// TIA Portal V17 export
// export: Created 2024-09-02T12:50:23.4161598Z, ExportSetting WithDefaults, DisplayName Totally Integrated Automation Portal, DisplayVersion V17, DisplayName TIA Portal Openness, DisplayVersion V17, DisplayName TIA Portal Version Control Interface, DisplayVersion V17, DisplayName STEP 7 Professional, DisplayVersion V17, DisplayName STEP 7 Safety, DisplayVersion V17, DisplayName WinCC Professional, DisplayVersion V17
FUNCTION "AnwFC_Aveva_OP702" : Void   // FC36, LAD
{ S7_Optimized_Access := 'TRUE' }
VERSION : 0.1
// stored: AutoNumber false, IsIECCheckEnabled false, SetENOAutomatically false, UDAEnableTagReadback false
   VAR_TEMP
      Data_Ready : Bool;
      Pallet_Nr_Moved : Bool;
      Converted_Data : Real;
      tEKSLevelOK : Bool;
   END_VAR
   VAR CONSTANT
      cButtonNotActive : USInt := 0;
      cButtonActive : USInt := 1;
      cColorRed : USInt := 2;
      cColorGreen : USInt := 3;
      cMesOptionEmpty : USInt := 0;
      cMesReasonEmpty : String := '';
   END_VAR
   VAR_TEMP   // added for the SCL form of the ladder/FBD networks
      _w1 : Bool;
      _w2 : Bool;
      _w3 : Bool;
      _w4 : Bool;
   END_VAR
BEGIN

REGION Network 1: ################STEP 1 - Pallet arrive to station #################
END_REGION

REGION Network 2: Copy Nr of Pallet
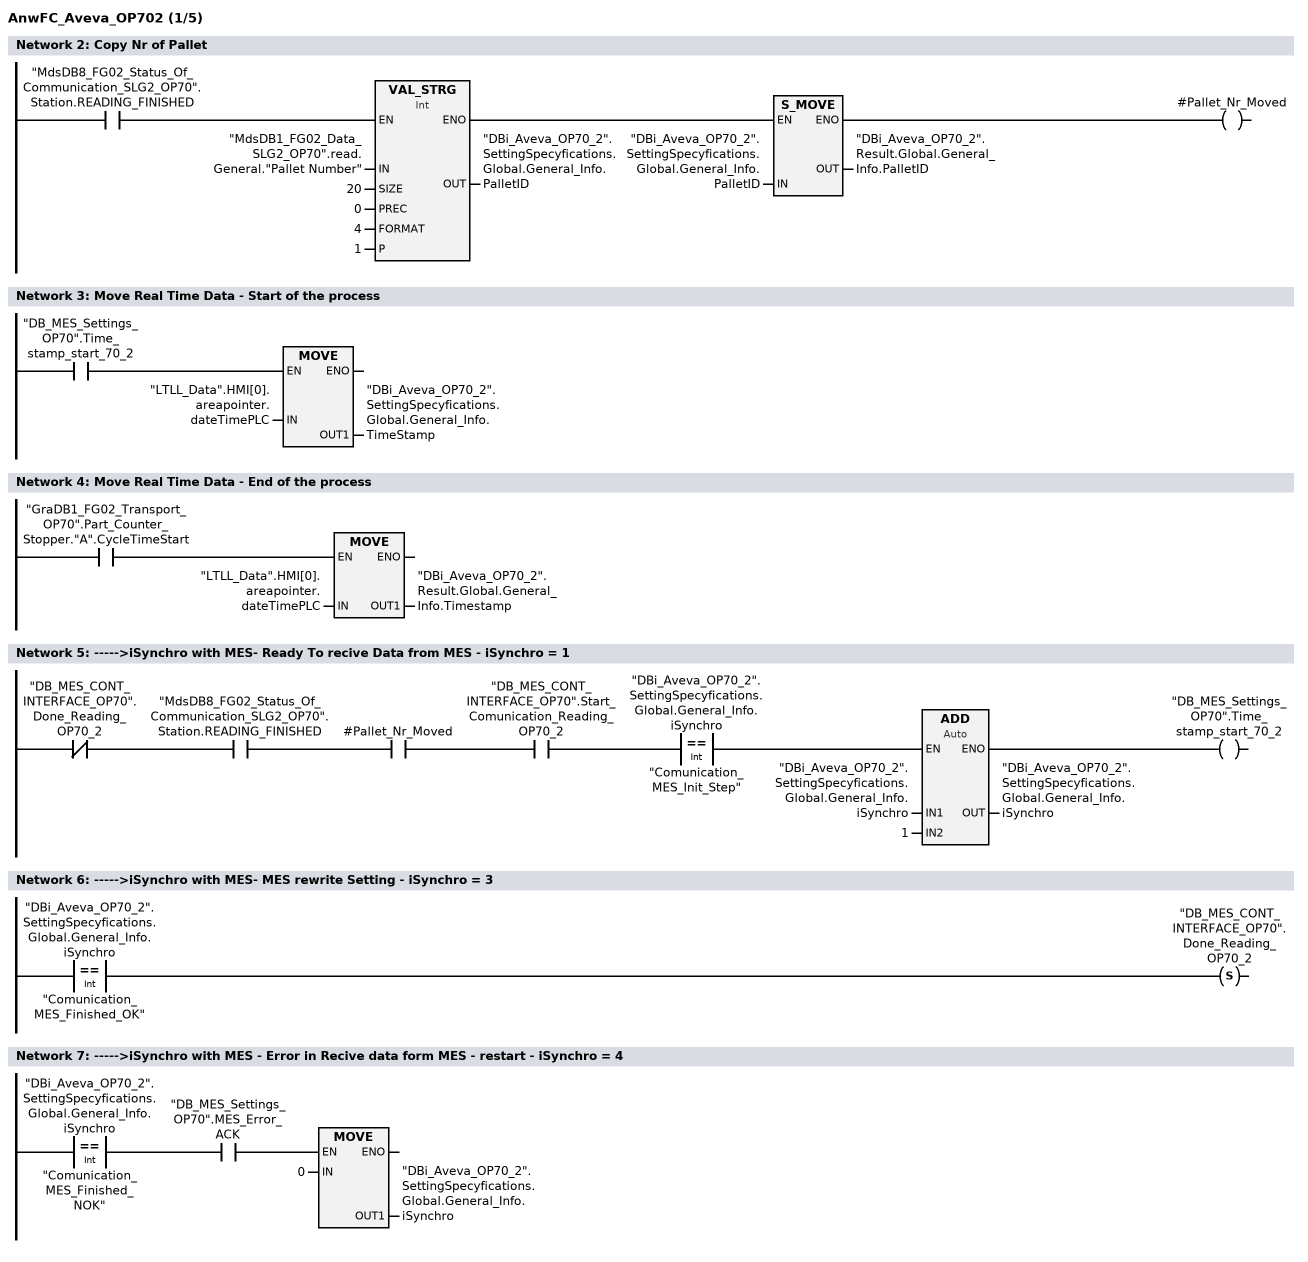
   RUNG wire#powerrail
      Contact( "MdsDB8_FG02_Status_Of_Communication_SLG2_OP70".Station.READING_FINISHED )
      { S7_Templates := "[value_type := Int, str_type := String]" } VAL_STRG(IN := "MdsDB1_FG02_Data_SLG2_OP70".read.General."Pallet Number", SIZE := 20, PREC := 0, FORMAT := 4, P := 1, OUT => "DBi_Aveva_OP70_2".SettingSpecyfications.Global.General_Info.PalletID)
      S_Move(in := "DBi_Aveva_OP70_2".SettingSpecyfications.Global.General_Info.PalletID, out => "DBi_Aveva_OP70_2".Result.Global.General_Info.PalletID)
      Coil( #Pallet_Nr_Moved )
   END_RUNG
   // the same network as SCL:
   VAL_STRG(EN := "MdsDB8_FG02_Status_Of_Communication_SLG2_OP70".Station.READING_FINISHED,
            IN := "MdsDB1_FG02_Data_SLG2_OP70".read.General."Pallet Number",
            SIZE := 20,
            PREC := 0,
            FORMAT := 4,
            P := 1,
            OUT => "DBi_Aveva_OP70_2".SettingSpecyfications.Global.General_Info.PalletID,
            ENO => #_w1);
   IF #_w1 THEN
       "DBi_Aveva_OP70_2".Result.Global.General_Info.PalletID := "DBi_Aveva_OP70_2".SettingSpecyfications.Global.General_Info.PalletID;
   END_IF;
   #Pallet_Nr_Moved := #_w1;
END_REGION

REGION Network 3: Move Real Time Data - Start of the process
   RUNG wire#powerrail
      Contact( "DB_MES_Settings_OP70".Time_stamp_start_70_2 )
      Move(in := "LTLL_Data".HMI[0].areapointer.dateTimePLC, out1 => "DBi_Aveva_OP70_2".SettingSpecyfications.Global.General_Info.TimeStamp)
   END_RUNG
   // the same network as SCL:
   IF "DB_MES_Settings_OP70".Time_stamp_start_70_2 THEN
       "DBi_Aveva_OP70_2".SettingSpecyfications.Global.General_Info.TimeStamp := "LTLL_Data".HMI[0].areapointer.dateTimePLC;
   END_IF;
END_REGION

REGION Network 4: Move Real Time Data - End of the process
   RUNG wire#powerrail
      Contact( "GraDB1_FG02_Transport_OP70".Part_Counter_Stopper."A".CycleTimeStart )
      Move(in := "LTLL_Data".HMI[0].areapointer.dateTimePLC, out1 => "DBi_Aveva_OP70_2".Result.Global.General_Info.Timestamp)
   END_RUNG
   // the same network as SCL:
   IF "GraDB1_FG02_Transport_OP70".Part_Counter_Stopper."A".CycleTimeStart THEN
       "DBi_Aveva_OP70_2".Result.Global.General_Info.Timestamp := "LTLL_Data".HMI[0].areapointer.dateTimePLC;
   END_IF;
END_REGION

REGION Network 5: ----->iSynchro with MES- Ready To recive Data from MES - iSynchro = 1
   RUNG wire#powerrail
      I_Contact( "DB_MES_CONT_INTERFACE_OP70".Done_Reading_OP70_2 )
      Contact( "MdsDB8_FG02_Status_Of_Communication_SLG2_OP70".Station.READING_FINISHED )
      Contact( #Pallet_Nr_Moved )
      Contact( "DB_MES_CONT_INTERFACE_OP70".Start_Comunication_Reading_OP70_2 )
      { S7_Templates := "SrcType := Int" } EQ_Contact(in1 := "DBi_Aveva_OP70_2".SettingSpecyfications.Global.General_Info.iSynchro, in2 := "Comunication_MES_Init_Step")
      Add(in1 := "DBi_Aveva_OP70_2".SettingSpecyfications.Global.General_Info.iSynchro, in2 := 1, out => "DBi_Aveva_OP70_2".SettingSpecyfications.Global.General_Info.iSynchro)
      Coil( "DB_MES_Settings_OP70".Time_stamp_start_70_2 )
   END_RUNG
   // the same network as SCL:
   #_w1 := NOT "DB_MES_CONT_INTERFACE_OP70".Done_Reading_OP70_2 AND "MdsDB8_FG02_Status_Of_Communication_SLG2_OP70".Station.READING_FINISHED AND #Pallet_Nr_Moved AND "DB_MES_CONT_INTERFACE_OP70".Start_Comunication_Reading_OP70_2 AND ("DBi_Aveva_OP70_2".SettingSpecyfications.Global.General_Info.iSynchro = "Comunication_MES_Init_Step");
   IF #_w1 THEN
       "DBi_Aveva_OP70_2".SettingSpecyfications.Global.General_Info.iSynchro := "DBi_Aveva_OP70_2".SettingSpecyfications.Global.General_Info.iSynchro + 1;
   END_IF;
   "DB_MES_Settings_OP70".Time_stamp_start_70_2 := #_w1;
END_REGION

REGION Network 6: ----->iSynchro with MES- MES rewrite Setting - iSynchro = 3
   RUNG wire#powerrail
      { S7_Templates := "SrcType := Int" } EQ_Contact(in1 := "DBi_Aveva_OP70_2".SettingSpecyfications.Global.General_Info.iSynchro, in2 := "Comunication_MES_Finished_OK")
      S_Coil( "DB_MES_CONT_INTERFACE_OP70".Done_Reading_OP70_2 )
   END_RUNG
   // the same network as SCL:
   IF "DBi_Aveva_OP70_2".SettingSpecyfications.Global.General_Info.iSynchro = "Comunication_MES_Finished_OK" THEN
       "DB_MES_CONT_INTERFACE_OP70".Done_Reading_OP70_2 := TRUE;
   END_IF;
END_REGION

REGION Network 7: ----->iSynchro with MES - Error in Recive data form MES - restart - iSynchro = 4
   RUNG wire#powerrail
      { S7_Templates := "SrcType := Int" } EQ_Contact(in1 := "DBi_Aveva_OP70_2".SettingSpecyfications.Global.General_Info.iSynchro, in2 := "Comunication_MES_Finished_NOK")
      Contact( "DB_MES_Settings_OP70".MES_Error_ACK )
      Move(in := 0, out1 => "DBi_Aveva_OP70_2".SettingSpecyfications.Global.General_Info.iSynchro)
   END_RUNG
   // the same network as SCL:
   IF ("DBi_Aveva_OP70_2".SettingSpecyfications.Global.General_Info.iSynchro = "Comunication_MES_Finished_NOK") AND "DB_MES_Settings_OP70".MES_Error_ACK THEN
       "DBi_Aveva_OP70_2".SettingSpecyfications.Global.General_Info.iSynchro := 0;
   END_IF;
END_REGION

REGION Network 8: ----->iSynchro with MES - End of Analyse - restart iSynchro = 0
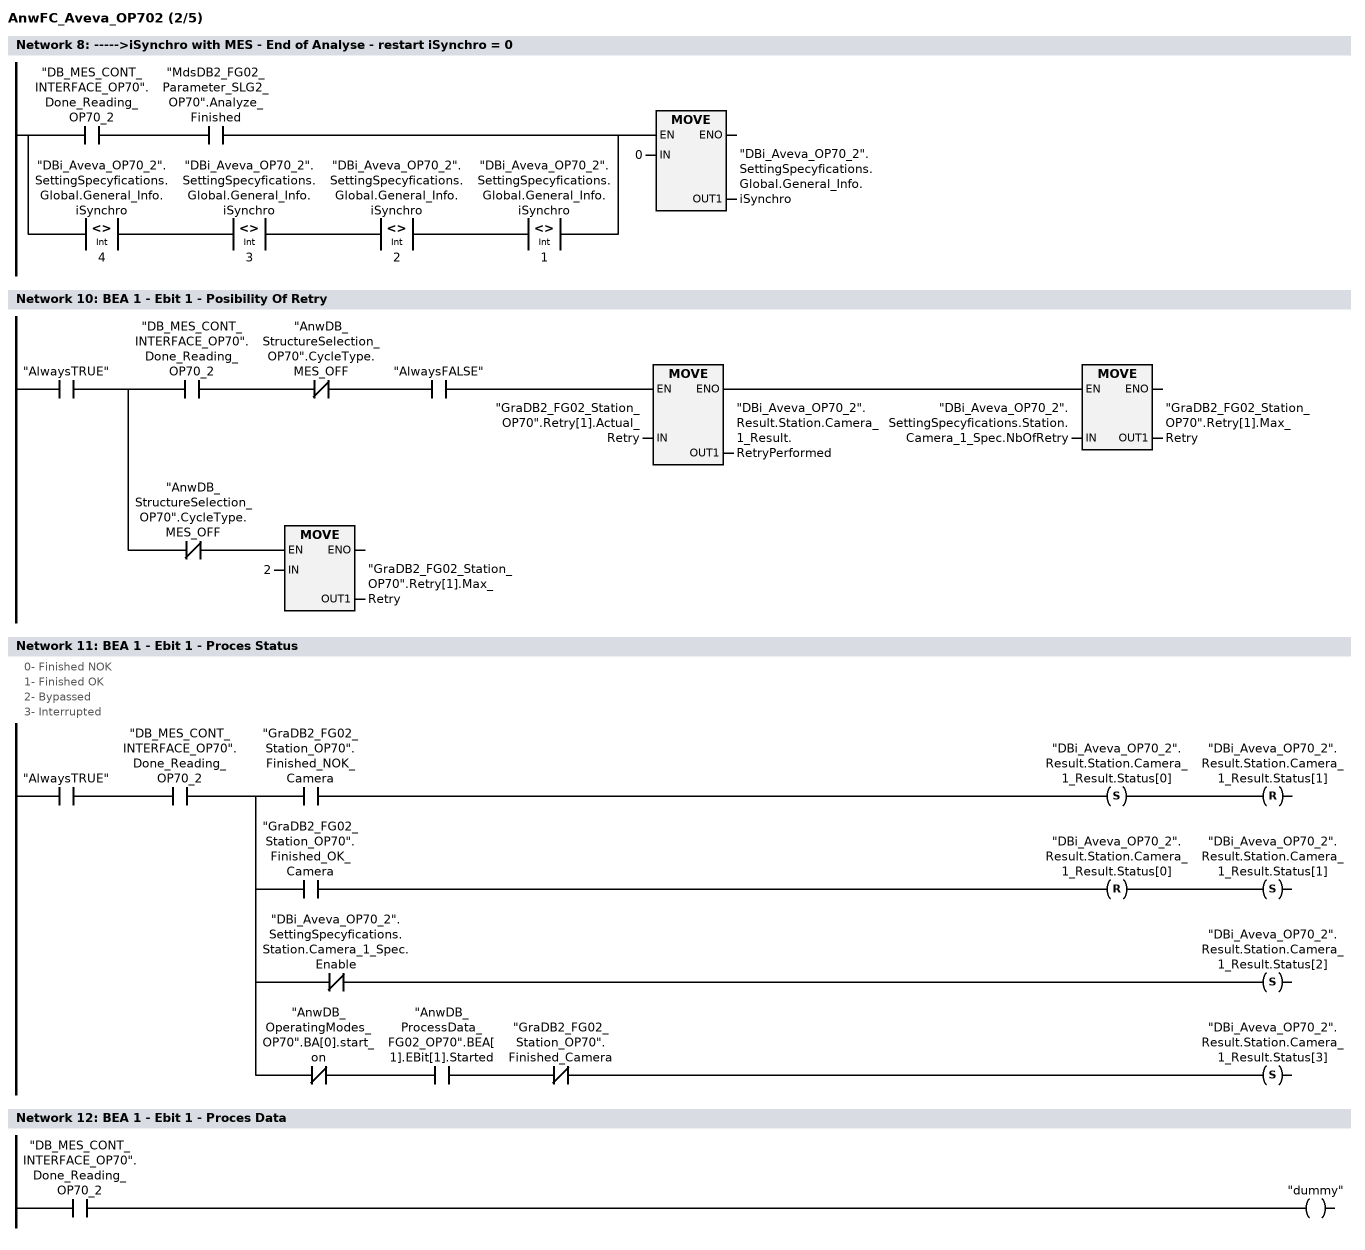
   RUNG wire#powerrail
      Contact( "DB_MES_CONT_INTERFACE_OP70".Done_Reading_OP70_2 )
      Contact( "MdsDB2_FG02_Parameter_SLG2_OP70".Analyze_Finished )
      wire#w1
      Move(in := 0, out1 => "DBi_Aveva_OP70_2".SettingSpecyfications.Global.General_Info.iSynchro)
   END_RUNG
   RUNG wire#powerrail
      { S7_Templates := "SrcType := Int" } NE_Contact(in1 := "DBi_Aveva_OP70_2".SettingSpecyfications.Global.General_Info.iSynchro, in2 := 4)
      { S7_Templates := "SrcType := Int" } NE_Contact(in1 := "DBi_Aveva_OP70_2".SettingSpecyfications.Global.General_Info.iSynchro, in2 := 3)
      { S7_Templates := "SrcType := Int" } NE_Contact(in1 := "DBi_Aveva_OP70_2".SettingSpecyfications.Global.General_Info.iSynchro, in2 := 2)
      { S7_Templates := "SrcType := Int" } NE_Contact(in1 := "DBi_Aveva_OP70_2".SettingSpecyfications.Global.General_Info.iSynchro, in2 := 1)
   END_RUNG wire#w1
   // the same network as SCL:
   IF ("DB_MES_CONT_INTERFACE_OP70".Done_Reading_OP70_2 AND "MdsDB2_FG02_Parameter_SLG2_OP70".Analyze_Finished) OR (("DBi_Aveva_OP70_2".SettingSpecyfications.Global.General_Info.iSynchro <> 4) AND ("DBi_Aveva_OP70_2".SettingSpecyfications.Global.General_Info.iSynchro <> 3) AND ("DBi_Aveva_OP70_2".SettingSpecyfications.Global.General_Info.iSynchro <> 2) AND ("DBi_Aveva_OP70_2".SettingSpecyfications.Global.General_Info.iSynchro <> 1)) THEN
       "DBi_Aveva_OP70_2".SettingSpecyfications.Global.General_Info.iSynchro := 0;
   END_IF;
END_REGION

REGION Network 9: ################STEP 2 - Move the Proce Data From Each Operation ################# / Status Proces 1
   // IN0 - Aktor ist abgewählt
   // IN1 - TAF ist angewählt
   // IN2 - Nacharbeit in Station
   // IN3 - Auftrag manuell vorgegeben
   // IN4 - Nacharbeit auf Standby-Platz
   // IN5 - Nacharbeit auf EAS-Platz
   // IN6 - TAF hat gearbeitet (Fertigmeldung)
   // IN7 - Bauteil wurde iO bearbeitet
END_REGION

REGION Network 10: BEA 1 - Ebit 1 - Posibility Of Retry
   RUNG wire#powerrail
      Contact( "AlwaysTRUE" )
      wire#w1
      Contact( "DB_MES_CONT_INTERFACE_OP70".Done_Reading_OP70_2 )
      I_Contact( "AnwDB_StructureSelection_OP70".CycleType.MES_OFF )
      Contact( "AlwaysFALSE" )
      Move(in := "GraDB2_FG02_Station_OP70".Retry[1].Actual_Retry, out1 => "DBi_Aveva_OP70_2".Result.Station.Camera_1_Result.RetryPerformed)
      Move(in := "DBi_Aveva_OP70_2".SettingSpecyfications.Station.Camera_1_Spec.NbOfRetry, out1 => "GraDB2_FG02_Station_OP70".Retry[1].Max_Retry)
   END_RUNG
   RUNG wire#w1
      I_Contact( "AnwDB_StructureSelection_OP70".CycleType.MES_OFF )
      Move(in := 2, out1 => "GraDB2_FG02_Station_OP70".Retry[1].Max_Retry)
   END_RUNG
   // the same network as SCL:
   IF "AlwaysTRUE" AND "DB_MES_CONT_INTERFACE_OP70".Done_Reading_OP70_2 AND NOT "AnwDB_StructureSelection_OP70".CycleType.MES_OFF AND "AlwaysFALSE" THEN
       "DBi_Aveva_OP70_2".Result.Station.Camera_1_Result.RetryPerformed := "GraDB2_FG02_Station_OP70".Retry[1].Actual_Retry;
       "GraDB2_FG02_Station_OP70".Retry[1].Max_Retry := "DBi_Aveva_OP70_2".SettingSpecyfications.Station.Camera_1_Spec.NbOfRetry;
   END_IF;
   IF "AlwaysTRUE" AND NOT "AnwDB_StructureSelection_OP70".CycleType.MES_OFF THEN
       "GraDB2_FG02_Station_OP70".Retry[1].Max_Retry := 2;
   END_IF;
END_REGION

REGION Network 11: BEA 1 - Ebit 1 - Proces Status
   // 0- Finished NOK
   // 1- Finished OK
   // 2- Bypassed
   // 3- Interrupted
   RUNG wire#powerrail
      Contact( "AlwaysTRUE" )
      Contact( "DB_MES_CONT_INTERFACE_OP70".Done_Reading_OP70_2 )
      wire#w1
      Contact( "GraDB2_FG02_Station_OP70".Finished_NOK_Camera )
      S_Coil( "DBi_Aveva_OP70_2".Result.Station.Camera_1_Result.Status[0] )
      R_Coil( "DBi_Aveva_OP70_2".Result.Station.Camera_1_Result.Status[1] )
   END_RUNG
   RUNG wire#w1
      Contact( "GraDB2_FG02_Station_OP70".Finished_OK_Camera )
      R_Coil( "DBi_Aveva_OP70_2".Result.Station.Camera_1_Result.Status[0] )
      S_Coil( "DBi_Aveva_OP70_2".Result.Station.Camera_1_Result.Status[1] )
   END_RUNG
   RUNG wire#w1
      I_Contact( "DBi_Aveva_OP70_2".SettingSpecyfications.Station.Camera_1_Spec.Enable )
      S_Coil( "DBi_Aveva_OP70_2".Result.Station.Camera_1_Result.Status[2] )
   END_RUNG
   RUNG wire#w1
      I_Contact( "AnwDB_OperatingModes_OP70".BA[0].start_on )
      Contact( "AnwDB_ProcessData_FG02_OP70".BEA[1].EBit[1].Started )
      I_Contact( "GraDB2_FG02_Station_OP70".Finished_Camera )
      S_Coil( "DBi_Aveva_OP70_2".Result.Station.Camera_1_Result.Status[3] )
   END_RUNG
   // the same network as SCL:
   #_w1 := "AlwaysTRUE" AND "DB_MES_CONT_INTERFACE_OP70".Done_Reading_OP70_2;
   IF #_w1 AND "GraDB2_FG02_Station_OP70".Finished_NOK_Camera THEN
       "DBi_Aveva_OP70_2".Result.Station.Camera_1_Result.Status[0] := TRUE;
       "DBi_Aveva_OP70_2".Result.Station.Camera_1_Result.Status[1] := FALSE;
   END_IF;
   IF #_w1 AND "GraDB2_FG02_Station_OP70".Finished_OK_Camera THEN
       "DBi_Aveva_OP70_2".Result.Station.Camera_1_Result.Status[0] := FALSE;
       "DBi_Aveva_OP70_2".Result.Station.Camera_1_Result.Status[1] := TRUE;
   END_IF;
   IF #_w1 AND NOT "DBi_Aveva_OP70_2".SettingSpecyfications.Station.Camera_1_Spec.Enable THEN
       "DBi_Aveva_OP70_2".Result.Station.Camera_1_Result.Status[2] := TRUE;
   END_IF;
   IF #_w1 AND NOT "AnwDB_OperatingModes_OP70".BA[0].start_on AND "AnwDB_ProcessData_FG02_OP70".BEA[1].EBit[1].Started AND NOT "GraDB2_FG02_Station_OP70".Finished_Camera THEN
       "DBi_Aveva_OP70_2".Result.Station.Camera_1_Result.Status[3] := TRUE;
   END_IF;
END_REGION

REGION Network 12: BEA 1 - Ebit 1 - Proces Data
   RUNG wire#powerrail
      Contact( "DB_MES_CONT_INTERFACE_OP70".Done_Reading_OP70_2 )
      Coil( "dummy" )
   END_RUNG
   // the same network as SCL:
   "dummy" := "DB_MES_CONT_INTERFACE_OP70".Done_Reading_OP70_2;
END_REGION

REGION Network 13: ------------------------------------------------------------
END_REGION

REGION Network 14: ################STEP 2 - Move the Proce Data From Station ################# / Status Proces 1
   // IN0 - Aktor ist abgewählt
   // IN1 - TAF ist angewählt
   // IN2 - Nacharbeit in Station
   // IN3 - Auftrag manuell vorgegeben
   // IN4 - Nacharbeit auf Standby-Platz
   // IN5 - Nacharbeit auf EAS-Platz
   // IN6 - TAF hat gearbeitet (Fertigmeldung)
   // IN7 - Bauteil wurde iO bearbeitet
END_REGION

REGION Network 15: Global Status of Station
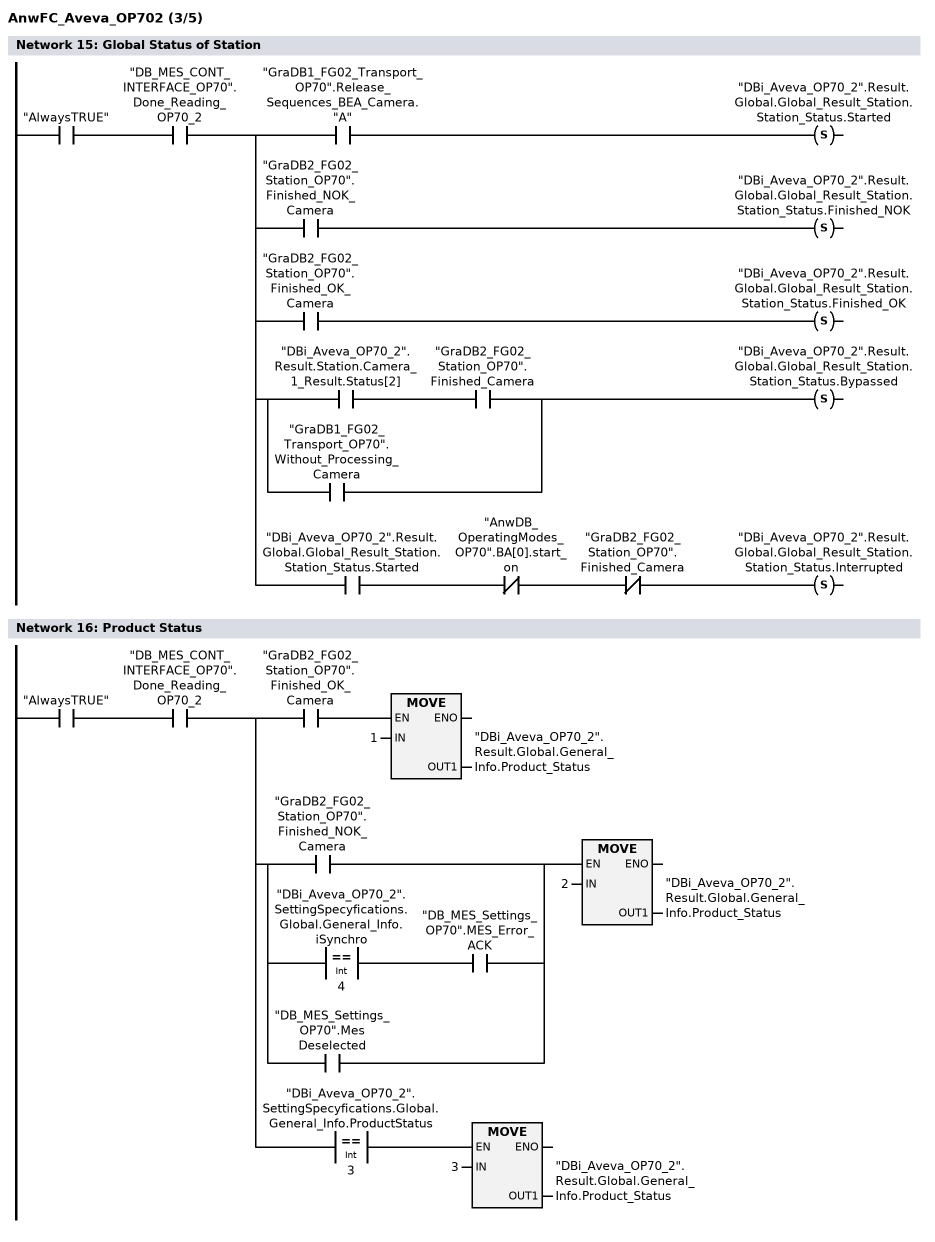
   RUNG wire#powerrail
      Contact( "AlwaysTRUE" )
      Contact( "DB_MES_CONT_INTERFACE_OP70".Done_Reading_OP70_2 )
      wire#w1
      Contact( "GraDB1_FG02_Transport_OP70".Release_Sequences_BEA_Camera."A" )
      S_Coil( "DBi_Aveva_OP70_2".Result.Global.Global_Result_Station.Station_Status.Started )
   END_RUNG
   RUNG wire#w1
      Contact( "GraDB2_FG02_Station_OP70".Finished_NOK_Camera )
      S_Coil( "DBi_Aveva_OP70_2".Result.Global.Global_Result_Station.Station_Status.Finished_NOK )
   END_RUNG
   RUNG wire#w1
      Contact( "GraDB2_FG02_Station_OP70".Finished_OK_Camera )
      S_Coil( "DBi_Aveva_OP70_2".Result.Global.Global_Result_Station.Station_Status.Finished_OK )
   END_RUNG
   RUNG wire#w1
      Contact( "DBi_Aveva_OP70_2".Result.Station.Camera_1_Result.Status[2] )
      Contact( "GraDB2_FG02_Station_OP70".Finished_Camera )
      wire#w2
      S_Coil( "DBi_Aveva_OP70_2".Result.Global.Global_Result_Station.Station_Status.Bypassed )
   END_RUNG
   RUNG wire#w1
      Contact( "GraDB1_FG02_Transport_OP70".Without_Processing_Camera )
   END_RUNG wire#w2
   RUNG wire#w1
      Contact( "DBi_Aveva_OP70_2".Result.Global.Global_Result_Station.Station_Status.Started )
      I_Contact( "AnwDB_OperatingModes_OP70".BA[0].start_on )
      I_Contact( "GraDB2_FG02_Station_OP70".Finished_Camera )
      S_Coil( "DBi_Aveva_OP70_2".Result.Global.Global_Result_Station.Station_Status.Interrupted )
   END_RUNG
   // the same network as SCL:
   #_w1 := "AlwaysTRUE" AND "DB_MES_CONT_INTERFACE_OP70".Done_Reading_OP70_2;
   IF #_w1 AND "GraDB1_FG02_Transport_OP70".Release_Sequences_BEA_Camera."A" THEN
       "DBi_Aveva_OP70_2".Result.Global.Global_Result_Station.Station_Status.Started := TRUE;
   END_IF;
   IF #_w1 AND "GraDB2_FG02_Station_OP70".Finished_NOK_Camera THEN
       "DBi_Aveva_OP70_2".Result.Global.Global_Result_Station.Station_Status.Finished_NOK := TRUE;
   END_IF;
   IF #_w1 AND "GraDB2_FG02_Station_OP70".Finished_OK_Camera THEN
       "DBi_Aveva_OP70_2".Result.Global.Global_Result_Station.Station_Status.Finished_OK := TRUE;
   END_IF;
   IF #_w1 AND (("DBi_Aveva_OP70_2".Result.Station.Camera_1_Result.Status[2] AND "GraDB2_FG02_Station_OP70".Finished_Camera) OR "GraDB1_FG02_Transport_OP70".Without_Processing_Camera) THEN
       "DBi_Aveva_OP70_2".Result.Global.Global_Result_Station.Station_Status.Bypassed := TRUE;
   END_IF;
   IF #_w1 AND "DBi_Aveva_OP70_2".Result.Global.Global_Result_Station.Station_Status.Started AND NOT "AnwDB_OperatingModes_OP70".BA[0].start_on AND NOT "GraDB2_FG02_Station_OP70".Finished_Camera THEN
       "DBi_Aveva_OP70_2".Result.Global.Global_Result_Station.Station_Status.Interrupted := TRUE;
   END_IF;
END_REGION

REGION Network 16: Product Status
   RUNG wire#powerrail
      Contact( "AlwaysTRUE" )
      Contact( "DB_MES_CONT_INTERFACE_OP70".Done_Reading_OP70_2 )
      wire#w1
      Contact( "GraDB2_FG02_Station_OP70".Finished_OK_Camera )
      Move(in := 1, out1 => "DBi_Aveva_OP70_2".Result.Global.General_Info.Product_Status)
   END_RUNG
   RUNG wire#w1
      Contact( "GraDB2_FG02_Station_OP70".Finished_NOK_Camera )
      wire#w2
      Move(in := 2, out1 => "DBi_Aveva_OP70_2".Result.Global.General_Info.Product_Status)
   END_RUNG
   RUNG wire#w1
      { S7_Templates := "SrcType := Int" } EQ_Contact(in1 := "DBi_Aveva_OP70_2".SettingSpecyfications.Global.General_Info.iSynchro, in2 := 4)
      Contact( "DB_MES_Settings_OP70".MES_Error_ACK )
   END_RUNG wire#w2
   RUNG wire#w1
      Contact( "DB_MES_Settings_OP70".MesDeselected )
   END_RUNG wire#w2
   RUNG wire#w1
      { S7_Templates := "SrcType := Int" } EQ_Contact(in1 := "DBi_Aveva_OP70_2".SettingSpecyfications.Global.General_Info.ProductStatus, in2 := 3)
      Move(in := 3, out1 => "DBi_Aveva_OP70_2".Result.Global.General_Info.Product_Status)
   END_RUNG
   // the same network as SCL:
   #_w1 := "AlwaysTRUE" AND "DB_MES_CONT_INTERFACE_OP70".Done_Reading_OP70_2;
   IF #_w1 AND "GraDB2_FG02_Station_OP70".Finished_OK_Camera THEN
       "DBi_Aveva_OP70_2".Result.Global.General_Info.Product_Status := 1;
   END_IF;
   IF #_w1 AND ("GraDB2_FG02_Station_OP70".Finished_NOK_Camera OR (("DBi_Aveva_OP70_2".SettingSpecyfications.Global.General_Info.iSynchro = 4) AND "DB_MES_Settings_OP70".MES_Error_ACK) OR "DB_MES_Settings_OP70".MesDeselected) THEN
       "DBi_Aveva_OP70_2".Result.Global.General_Info.Product_Status := 2;
   END_IF;
   IF #_w1 AND ("DBi_Aveva_OP70_2".SettingSpecyfications.Global.General_Info.ProductStatus = 3) THEN
       "DBi_Aveva_OP70_2".Result.Global.General_Info.Product_Status := 3;
   END_IF;
END_REGION

REGION Network 17: ################ STEP 3 - Prepare Isynchro for MES in result area #################
END_REGION

REGION Network 18: ----->iSynchro with MES- Ready To copy Data to MES - iSynchro = 1
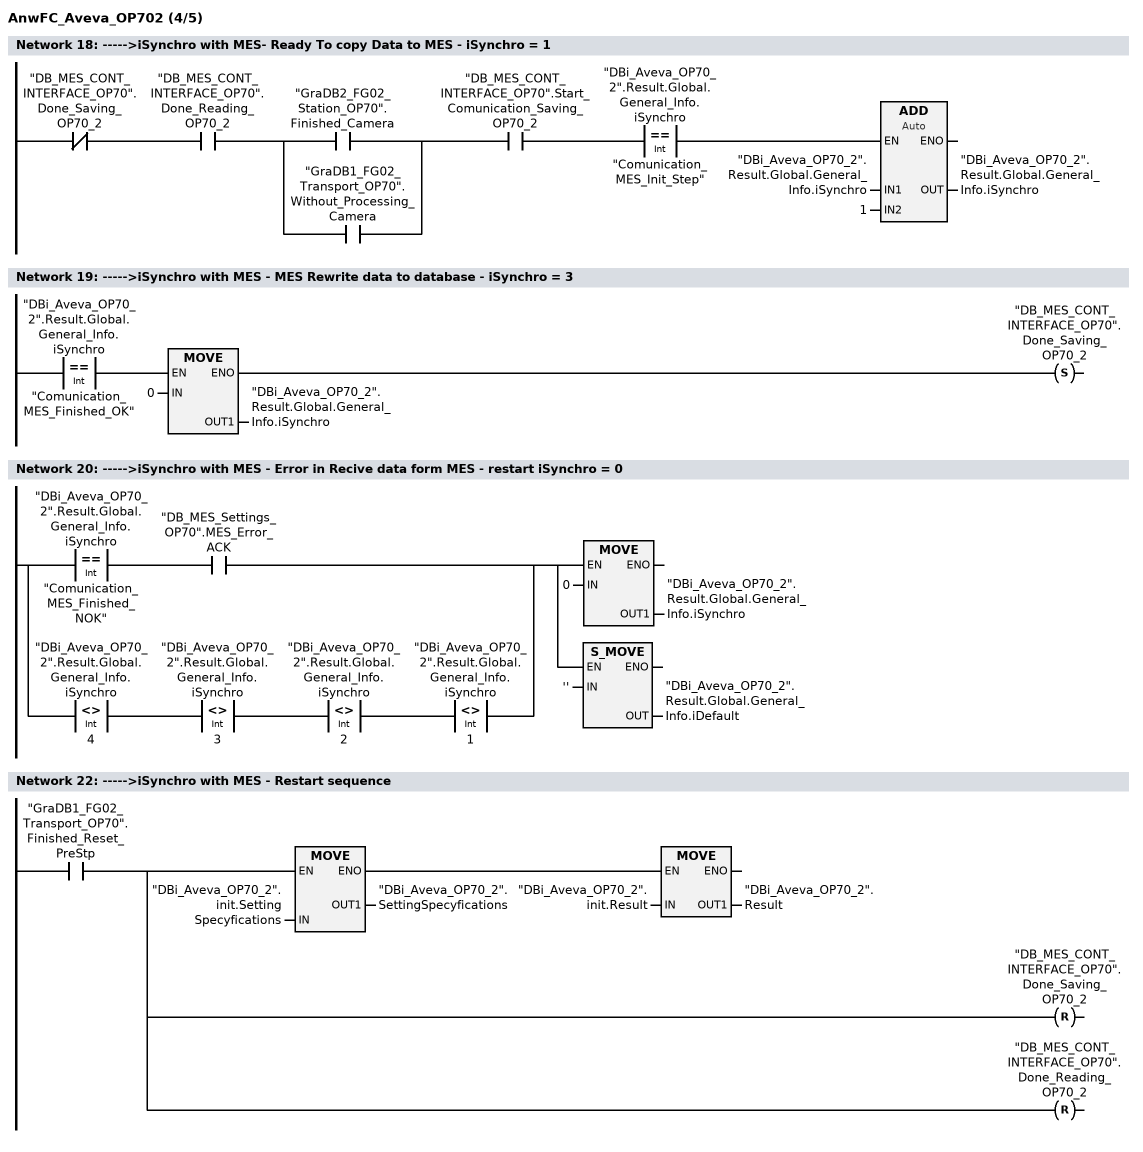
   RUNG wire#powerrail
      I_Contact( "DB_MES_CONT_INTERFACE_OP70".Done_Saving_OP70_2 )
      Contact( "DB_MES_CONT_INTERFACE_OP70".Done_Reading_OP70_2 )
      wire#w1
      Contact( "GraDB2_FG02_Station_OP70".Finished_Camera )
      wire#w2
      Contact( "DB_MES_CONT_INTERFACE_OP70".Start_Comunication_Saving_OP70_2 )
      { S7_Templates := "SrcType := Int" } EQ_Contact(in1 := "DBi_Aveva_OP70_2".Result.Global.General_Info.iSynchro, in2 := "Comunication_MES_Init_Step")
      Add(in1 := "DBi_Aveva_OP70_2".Result.Global.General_Info.iSynchro, in2 := 1, out => "DBi_Aveva_OP70_2".Result.Global.General_Info.iSynchro)
   END_RUNG
   RUNG wire#w1
      Contact( "GraDB1_FG02_Transport_OP70".Without_Processing_Camera )
   END_RUNG wire#w2
   // the same network as SCL:
   IF NOT "DB_MES_CONT_INTERFACE_OP70".Done_Saving_OP70_2 AND "DB_MES_CONT_INTERFACE_OP70".Done_Reading_OP70_2 AND ("GraDB2_FG02_Station_OP70".Finished_Camera OR "GraDB1_FG02_Transport_OP70".Without_Processing_Camera) AND "DB_MES_CONT_INTERFACE_OP70".Start_Comunication_Saving_OP70_2 AND ("DBi_Aveva_OP70_2".Result.Global.General_Info.iSynchro = "Comunication_MES_Init_Step") THEN
       "DBi_Aveva_OP70_2".Result.Global.General_Info.iSynchro := "DBi_Aveva_OP70_2".Result.Global.General_Info.iSynchro + 1;
   END_IF;
END_REGION

REGION Network 19: ----->iSynchro with MES - MES Rewrite data to database - iSynchro = 3
   RUNG wire#powerrail
      { S7_Templates := "SrcType := Int" } EQ_Contact(in1 := "DBi_Aveva_OP70_2".Result.Global.General_Info.iSynchro, in2 := "Comunication_MES_Finished_OK")
      Move(in := 0, out1 => "DBi_Aveva_OP70_2".Result.Global.General_Info.iSynchro)
      S_Coil( "DB_MES_CONT_INTERFACE_OP70".Done_Saving_OP70_2 )
   END_RUNG
   // the same network as SCL:
   #_w1 := "DBi_Aveva_OP70_2".Result.Global.General_Info.iSynchro = "Comunication_MES_Finished_OK";
   IF #_w1 THEN
       "DBi_Aveva_OP70_2".Result.Global.General_Info.iSynchro := 0;
       "DB_MES_CONT_INTERFACE_OP70".Done_Saving_OP70_2 := TRUE;
   END_IF;
END_REGION

REGION Network 20: ----->iSynchro with MES - Error in Recive data form MES - restart iSynchro = 0
   RUNG wire#powerrail
      { S7_Templates := "SrcType := Int" } EQ_Contact(in1 := "DBi_Aveva_OP70_2".Result.Global.General_Info.iSynchro, in2 := "Comunication_MES_Finished_NOK")
      Contact( "DB_MES_Settings_OP70".MES_Error_ACK )
      wire#w1
      Move(in := 0, out1 => "DBi_Aveva_OP70_2".Result.Global.General_Info.iSynchro)
   END_RUNG
   RUNG wire#powerrail
      { S7_Templates := "SrcType := Int" } NE_Contact(in1 := "DBi_Aveva_OP70_2".Result.Global.General_Info.iSynchro, in2 := 4)
      { S7_Templates := "SrcType := Int" } NE_Contact(in1 := "DBi_Aveva_OP70_2".Result.Global.General_Info.iSynchro, in2 := 3)
      { S7_Templates := "SrcType := Int" } NE_Contact(in1 := "DBi_Aveva_OP70_2".Result.Global.General_Info.iSynchro, in2 := 2)
      { S7_Templates := "SrcType := Int" } NE_Contact(in1 := "DBi_Aveva_OP70_2".Result.Global.General_Info.iSynchro, in2 := 1)
   END_RUNG wire#w1
   RUNG wire#w1
      S_Move(in := '', out => "DBi_Aveva_OP70_2".Result.Global.General_Info.iDefault)
   END_RUNG
   // the same network as SCL:
   #_w1 := (("DBi_Aveva_OP70_2".Result.Global.General_Info.iSynchro = "Comunication_MES_Finished_NOK") AND "DB_MES_Settings_OP70".MES_Error_ACK) OR (("DBi_Aveva_OP70_2".Result.Global.General_Info.iSynchro <> 4) AND ("DBi_Aveva_OP70_2".Result.Global.General_Info.iSynchro <> 3) AND ("DBi_Aveva_OP70_2".Result.Global.General_Info.iSynchro <> 2) AND ("DBi_Aveva_OP70_2".Result.Global.General_Info.iSynchro <> 1));
   IF #_w1 THEN
       "DBi_Aveva_OP70_2".Result.Global.General_Info.iSynchro := 0;
       "DBi_Aveva_OP70_2".Result.Global.General_Info.iDefault := '';
   END_IF;
END_REGION

REGION Network 21: ################ STEP3 - Restart all #################
END_REGION

REGION Network 22: ----->iSynchro with MES - Restart sequence
   RUNG wire#powerrail
      Contact( "GraDB1_FG02_Transport_OP70".Finished_Reset_PreStp )
      wire#w1
      Move(in := "DBi_Aveva_OP70_2".init.SettingSpecyfications, out1 => "DBi_Aveva_OP70_2".SettingSpecyfications)
      Move(in := "DBi_Aveva_OP70_2".init.Result, out1 => "DBi_Aveva_OP70_2".Result)
   END_RUNG
   RUNG wire#w1
      R_Coil( "DB_MES_CONT_INTERFACE_OP70".Done_Saving_OP70_2 )
   END_RUNG
   RUNG wire#w1
      R_Coil( "DB_MES_CONT_INTERFACE_OP70".Done_Reading_OP70_2 )
   END_RUNG
   // the same network as SCL:
   IF "GraDB1_FG02_Transport_OP70".Finished_Reset_PreStp THEN
       "DBi_Aveva_OP70_2".SettingSpecyfications := "DBi_Aveva_OP70_2".init.SettingSpecyfications;
       "DBi_Aveva_OP70_2".Result := "DBi_Aveva_OP70_2".init.Result;
       "DB_MES_CONT_INTERFACE_OP70".Done_Saving_OP70_2 := FALSE;
       "DB_MES_CONT_INTERFACE_OP70".Done_Reading_OP70_2 := FALSE;
   END_IF;
END_REGION

REGION Network 23: ################ Status of machine #################
END_REGION

REGION Network 24: Auto/ Hand/ Station started/ Error
   // %X0 - (WS)Media ON, 
   // %X1 - (WS)Hand selected,
   // %X2 - (WS)Auto selected, 
   // %X3 - (WS)Start ON(with auto or hand Mode),  
   // %X4 - (WS)Error,  
   // %X5 - (WS)Clock_1Hz - lifebit, 
   // %X6 - (MES)Clock_1Hz - lifebit ,  
   // %X7 - (MES)Automatic on Conveyor
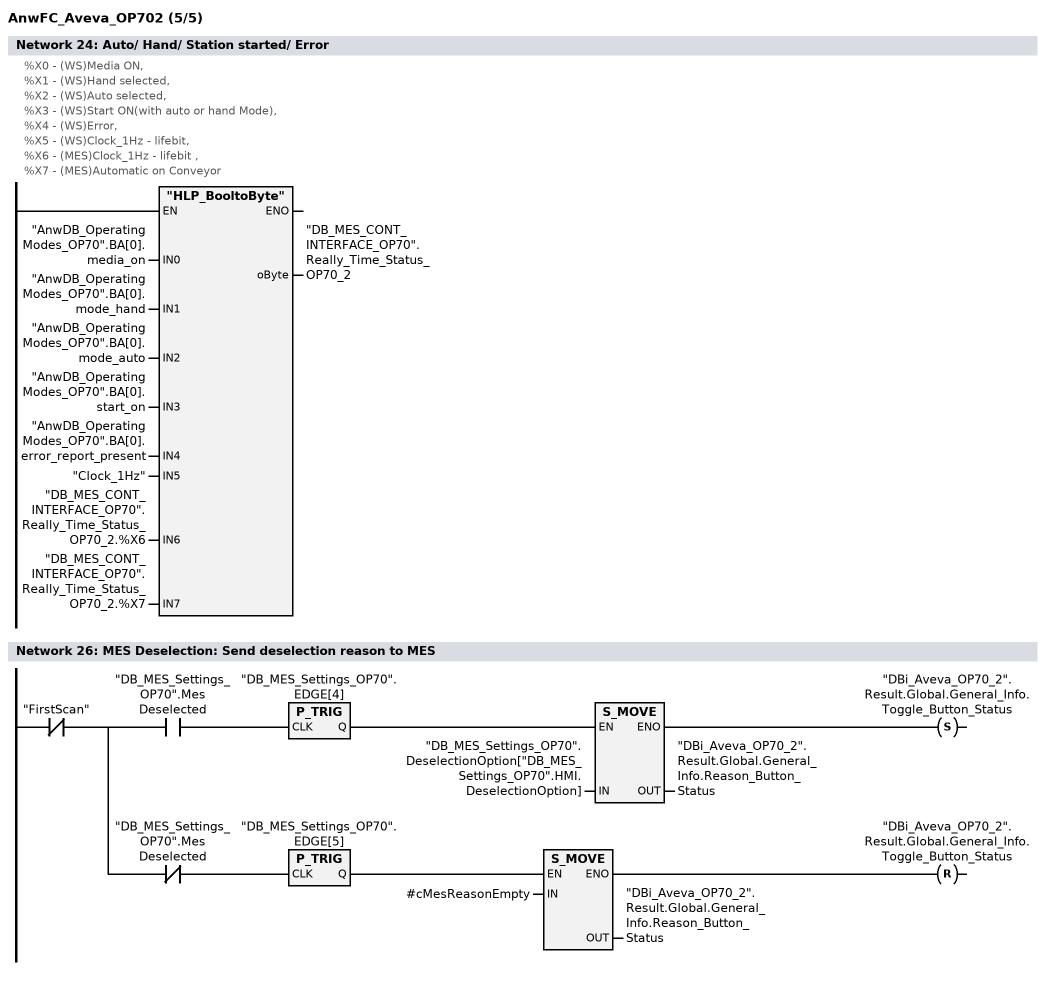
   RUNG wire#powerrail
      "HLP_BooltoByte"(IN0 := "AnwDB_OperatingModes_OP70".BA[0].media_on, IN1 := "AnwDB_OperatingModes_OP70".BA[0].mode_hand, IN2 := "AnwDB_OperatingModes_OP70".BA[0].mode_auto, IN3 := "AnwDB_OperatingModes_OP70".BA[0].start_on, IN4 := "AnwDB_OperatingModes_OP70".BA[0].error_report_present, IN5 := "Clock_1Hz", IN6 := "DB_MES_CONT_INTERFACE_OP70".Really_Time_Status_OP70_2.%X6, IN7 := "DB_MES_CONT_INTERFACE_OP70".Really_Time_Status_OP70_2.%X7, oByte => "DB_MES_CONT_INTERFACE_OP70".Really_Time_Status_OP70_2)
   END_RUNG
   // the same network as SCL:
   "HLP_BooltoByte"(IN0 := "AnwDB_OperatingModes_OP70".BA[0].media_on,
                    IN1 := "AnwDB_OperatingModes_OP70".BA[0].mode_hand,
                    IN2 := "AnwDB_OperatingModes_OP70".BA[0].mode_auto,
                    IN3 := "AnwDB_OperatingModes_OP70".BA[0].start_on,
                    IN4 := "AnwDB_OperatingModes_OP70".BA[0].error_report_present,
                    IN5 := "Clock_1Hz",
                    IN6 := "DB_MES_CONT_INTERFACE_OP70".Really_Time_Status_OP70_2.%X6,
                    IN7 := "DB_MES_CONT_INTERFACE_OP70".Really_Time_Status_OP70_2.%X7,
                    oByte => "DB_MES_CONT_INTERFACE_OP70".Really_Time_Status_OP70_2);
END_REGION

REGION Network 25: ################ MES DESELECTION #################
END_REGION

REGION Network 26: MES Deselection: Send deselection reason to MES
   RUNG wire#powerrail
      I_Contact( "FirstScan" )
      wire#w1
      Contact( "DB_MES_Settings_OP70".MesDeselected )
      P_Trig( "DB_MES_Settings_OP70".EDGE[4] )
      S_Move(in := "DB_MES_Settings_OP70".DeselectionOption["DB_MES_Settings_OP70".HMI.DeselectionOption], out => "DBi_Aveva_OP70_2".Result.Global.General_Info.Reason_Button_Status)
      S_Coil( "DBi_Aveva_OP70_2".Result.Global.General_Info.Toggle_Button_Status )
   END_RUNG
   RUNG wire#w1
      I_Contact( "DB_MES_Settings_OP70".MesDeselected )
      P_Trig( "DB_MES_Settings_OP70".EDGE[5] )
      S_Move(in := #cMesReasonEmpty, out => "DBi_Aveva_OP70_2".Result.Global.General_Info.Reason_Button_Status)
      R_Coil( "DBi_Aveva_OP70_2".Result.Global.General_Info.Toggle_Button_Status )
   END_RUNG
   // the same network as SCL:
   #_w1 := NOT "FirstScan" AND "DB_MES_Settings_OP70".MesDeselected;
   #_w2 := #_w1 AND NOT "DB_MES_Settings_OP70".EDGE[4];   // rising edge
   "DB_MES_Settings_OP70".EDGE[4] := #_w1;
   IF #_w2 THEN
       "DBi_Aveva_OP70_2".Result.Global.General_Info.Reason_Button_Status := "DB_MES_Settings_OP70".DeselectionOption["DB_MES_Settings_OP70".HMI.DeselectionOption];
       "DBi_Aveva_OP70_2".Result.Global.General_Info.Toggle_Button_Status := TRUE;
   END_IF;
   #_w3 := NOT "FirstScan" AND NOT "DB_MES_Settings_OP70".MesDeselected;
   #_w4 := #_w3 AND NOT "DB_MES_Settings_OP70".EDGE[5];   // rising edge
   "DB_MES_Settings_OP70".EDGE[5] := #_w3;
   IF #_w4 THEN
       "DBi_Aveva_OP70_2".Result.Global.General_Info.Reason_Button_Status := #cMesReasonEmpty;
       "DBi_Aveva_OP70_2".Result.Global.General_Info.Toggle_Button_Status := FALSE;
   END_IF;
END_REGION
END_FUNCTION
